(* CoDeSys 2.3.9.41 project: proj1.pro *)

(* POU PLC_PRG, ST *)
PROGRAM PLC_PRG
VAR
	x,y:INT;
END_VAR
x:=x+1;
y:=y+1;
END_PROGRAM
